FUNCTION_BLOCK DrillModelView
  (* Standard: 61499-2 *)
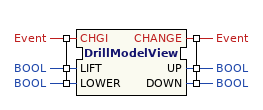
  EVENT_INPUT
    CHGI WITH LIFT, LOWER;
  END_EVENT
  EVENT_OUTPUT
    CHANGE WITH UP, DOWN;
  END_EVENT
  VAR_INPUT
    LIFT : BOOL;
    LOWER : BOOL;
  END_VAR
  VAR_OUTPUT
    UP : BOOL;
    DOWN : BOOL;
  END_VAR
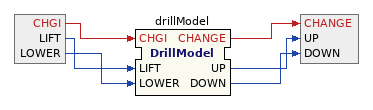
  FBS
    drillModel : DrillModel;
  END_FBS
  EVENT_CONNECTIONS
    CHGI TO drillModel.CHGI;
    drillModel.CHANGE TO CHANGE;
  END_CONNECTIONS
  DATA_CONNECTIONS
    LIFT TO drillModel.LIFT;
    LOWER TO drillModel.LOWER;
    drillModel.UP TO UP;
    drillModel.DOWN TO DOWN;
  END_CONNECTIONS
END_FUNCTION_BLOCK
